PROGRAM PRG_Section_2
VAR
END_VAR

END_PROGRAM

(* stored: Version 1.1.0.1, ProductVersion 3.1.4022.18
   POU PRG_Section_2: Id {aa241f3d-e544-47fe-9c03-27baee63cd5a}, SpecialFunc None *)
